(* IEC 61131-3 sources: ics/BLR1_PhoenixContact/BLR1_AXC1050_21/LogicalPOUs/MTR, 6 files *)

(* ---- MotorFB.ST ---- *)
(*@PROPERTIES_EX@
TYPE: POU
LOCALE: 0
IEC_LANGUAGE: ST
PLC_TYPE: independent
PROC_TYPE: independent
GROUP: MTRS.FB
*)
(*@KEY@:DESCRIPTION*)

(*@KEY@:END_DESCRIPTION*)
FUNCTION_BLOCK MotorFB

(*Group:Default*)

VAR_IN_OUT
    Mot_strct :	MTR;
    Aux_strct :	MTR_MISC;
END_VAR

VAR_INPUT
    Cycle :	CCL;
END_VAR

VAR_EXTERNAL
    TICK_1S_PLS :	BOOL;
END_VAR

VAR_OUTPUT
    Event :	MTR_EVENT;
END_VAR

(*@KEY@: WORKSHEET
NAME: MotorFB
IEC_LANGUAGE: ST
*)

IF TICK_1S_PLS and not Aux_strct.AuxFlag THEN
    Aux_strct.Tick_1S:= true;
END_IF;
Aux_strct.AuxFlag:= TICK_1S_PLS;

(*============================================================================*)
    (*Alarm Feedback processing*)
(*============================================================================*)
IF Mot_strct.CW.Enable and ((Aux_strct.COM and not Mot_strct.SW.RUN) or (not Aux_strct.COM and Mot_strct.SW.RUN)) THEN
    IF Aux_strct.Tick_1S THEN
        Aux_strct.AlrmTickCount:= Aux_strct.AlrmTickCount + 1;
    END_IF;
ELSE
    Aux_strct.AlrmTickCount:= 0;
END_IF;

IF Aux_strct.AlrmTickCount >= Aux_strct.SetOvertime THEN
    Aux_strct.AlarmFeedback:=true;
    Aux_strct.AlrmTickCount:= 0;
END_IF;

IF not Mot_strct.CW.ExtraEn and Aux_strct.COM THEN
    Aux_strct.AlarmBlock:= true;
END_IF;

Mot_strct.SW.AlarmAccum:= Aux_strct.AlarmFeedback or Mot_strct.CW.ExtraAlarm or Aux_strct.AlarmBlock;

IF Mot_strct.CW.ACK THEN
    Aux_strct.AlarmFeedback:=false;
    Aux_strct.AlarmBlock:= false;
END_IF;

(*============================================================================*)
    (*Auto/Manual mode selection*)
(*============================================================================*)
IF Mot_strct.CW.AutoMode THEN
    Mot_strct.SW.ManAuto:= true;
ELSIF Mot_strct.CW.ManMode THEN
    Mot_strct.SW.ManAuto:= false;
END_IF;

Mot_strct.SW.ManOK:= not Mot_strct.SW.AlarmAccum and Mot_strct.CW.AuxON and
    Mot_strct.CW.Enable and not Mot_strct.SW.ManAuto;
Mot_strct.SW.AutoOK:= not Mot_strct.SW.AlarmAccum and Mot_strct.CW.AuxON and
    Mot_strct.CW.Enable and Mot_strct.SW.ManAuto;

(*============================================================================*)
    (*Manual mode activation*)
(*============================================================================*)

IF Mot_strct.CW.ManStop or not Mot_strct.SW.ManOK THEN
    Mot_strct.SW.RunManual:=false;
ELSIF Mot_strct.CW.ManStart THEN
    Mot_strct.SW.RunManual:=true;
END_IF;

(*============================================================================*)
    (*Auto mode activation*)
(*============================================================================*)
Mot_strct.SW.RunAuto:= Mot_strct.SW.AutoOK and Cycle.SW.Running;

(*============================================================================*)
    (*Set command for start*)
(*============================================================================*)
Aux_strct.COM:=((Mot_strct.SW.RunManual and Mot_strct.SW.ManOK) or
    (Mot_strct.SW.RunAuto and Mot_strct.SW.AutoOK and Mot_strct.CW.AutoON));
Mot_strct.SW.COM:=Aux_strct.COM and not Mot_strct.CW.SimEn;

(*============================================================================*)
    (*Frequency limatation*)
(*============================================================================*)
Mot_strct.MaxFreq:= LIMIT(0.0, Mot_strct.MaxFreq, 50.0);
Mot_strct.MinFreq:= LIMIT(0.0, Mot_strct.MinFreq, Mot_strct.MaxFreq);
Mot_strct.ManFreq:= LIMIT(Mot_strct.MinFreq, Mot_strct.ManFreq, Mot_strct.MaxFreq);
Mot_strct.AutoFreq:= LIMIT(Mot_strct.MinFreq, Mot_strct.AutoFreq, Mot_strct.MaxFreq);

IF Mot_strct.SW.RunAuto and not Mot_strct.SW.AlarmAccum and Mot_strct.CW.AuxON THEN
    Aux_strct.SetValue:=Mot_strct.AutoFreq;
ELSIF not Mot_strct.SW.AlarmAccum and Mot_strct.SW.RunManual THEN
    Aux_strct.SetValue:=Mot_strct.ManFreq;
ELSE
    Aux_strct.SetValue:=0.0;
END_IF;

(*============================================================================*)
    (*Work time counter*)
(*============================================================================*)
IF Mot_strct.SW.COM and Aux_strct.Tick_1S THEN
    Aux_strct.Seconds:= Aux_strct.Seconds + udint#1;
END_IF;

Aux_strct.Minutes:= Aux_strct.Seconds / udint#60;
Aux_strct.Hours:= Aux_strct.Seconds / udint#3600;
Aux_strct.Days:= Aux_strct.Seconds / udint#86400;

(*============================================================================*)
    (*Aux time counters*)
(*============================================================================*)
IF Aux_strct.CT1_ON and Aux_strct.Tick_1S THEN
    Aux_strct.CT1:= Aux_strct.CT1 + 1;
ELSIF not Aux_strct.CT1_ON THEN
    Aux_strct.CT1:= 0;
END_IF;

IF Aux_strct.CT2_ON and Aux_strct.Tick_1S THEN
    Aux_strct.CT2:= Aux_strct.CT2 + 1;
ELSIF not Aux_strct.CT2_ON THEN
    Aux_strct.CT2:= 0;
END_IF;

(*============================================================================*)
    (*Status processing*)
(*============================================================================*)
IF Mot_strct.SW.AlarmAccum THEN                                                 (*Alarm*)
    Mot_strct.Status:=word#2;
ELSIF not Mot_strct.CW.ExtraEn THEN                                             (*Blocking*)
    Mot_strct.Status:=word#4;
ELSIF Mot_strct.SW.COM THEN                                                     (*Working*)
    Mot_strct.Status:=word#1;
ELSE                                                                            (*Stopped*)
    Mot_strct.Status:=word#0;
END_IF;

Mot_strct.CW.AutoMode:=false;
Mot_strct.CW.ManMode:=false;
Mot_strct.CW.ManStart:=false;
Mot_strct.CW.ManStop:=false;
Mot_strct.CW.ACK:=false;
Aux_strct.Tick_1S:= false;

(*============================================================================*)
(*Motor Pulse Events*)
(*============================================================================*)

Event.AlarmAccum:= false;
IF Mot_strct.SW.AlarmAccum and not Aux_strct.EVENT_1 THEN
    Event.AlarmAccum:= true;
    Aux_strct.EVENT_1:= true;
ELSIF not Mot_strct.SW.AlarmAccum THEN
    Aux_strct.EVENT_1:= false;
END_IF;
(*@KEY@: END_WORKSHEET *)
END_FUNCTION_BLOCK

(* ---- BLR_CTRL.ST ---- *)
(*@PROPERTIES_EX@
TYPE: POU
LOCALE: 0
IEC_LANGUAGE: ST
PLC_TYPE: independent
PROC_TYPE: independent
GROUP: MTRS
*)
(*@KEY@:DESCRIPTION*)

(*@KEY@:END_DESCRIPTION*)
PROGRAM BLR_CTRL

(*Group:Default*)

(*@KEY@: WORKSHEET
NAME: BLR_CTRL
IEC_LANGUAGE: ST
*)
(*@KEY@: END_WORKSHEET *)
END_PROGRAM

(* ---- MTR.ST ---- *)
(*@PROPERTIES_EX@
TYPE: POU
LOCALE: 0
IEC_LANGUAGE: ST
PLC_TYPE: independent
PROC_TYPE: independent
GROUP: MTRS
*)
(*@KEY@:DESCRIPTION*)

(*@KEY@:END_DESCRIPTION*)
PROGRAM MTR

(*Group:Default*)

VAR_EXTERNAL
    Cycle :	CCL;
    M :	MOTOR;
    WarnWord :	WRN;
    AI :	SENSOR;
END_VAR

VAR
    Pmp31FB :	MotorFB;
END_VAR

VAR_EXTERNAL
    M_AUX :	MOTOR_MISC;
END_VAR

VAR
    i :	INT;
    PmpsFB :	MotorFB;
END_VAR

VAR_EXTERNAL
    Blr11_BrnRun :	BOOL;
    Blr11_BrnFault :	BOOL;
    Blr12_BrnRun :	BOOL;
    Blr12_BrnFault :	BOOL;
    Blr13_BrnRun :	BOOL;
    Blr13_BrnFault :	BOOL;
    Blr21_BrnRun :	BOOL;
    Blr21_BrnFault :	BOOL;
    Blr22_BrnRun :	BOOL;
    Blr22_BrnFault :	BOOL;
END_VAR

VAR
    PumpsFB :	MotorFB;
    MB_TO_REAL :	MB_TO_REAL;
END_VAR

VAR_EXTERNAL
    SlvData_RSUNI_2 :	MBRTU_SlvData;
    SlvData_RSUNI_1 :	MBRTU_SlvData;
    MBTCP_Data :	MB_TCP_ARR_W_0_7167;
END_VAR

VAR
    j :	INT;
    j2 :	INT;
    j3 :	INT;
    j4 :	INT;
    j5 :	INT;
    j6 :	INT;
    j7 :	INT;
    REAL_TO_MB :	REAL_TO_MB;
    BoilersFB :	MotorFB;
    BlrCycle :	CCL;
END_VAR

VAR_EXTERNAL
    CCL :	CYCLE;
    Blr11_EmergCirc :	BOOL;
    Blr12_EmergCirc :	BOOL;
    Blr13_EmergCirc :	BOOL;
    Blr21_EmergCirc :	BOOL;
    Blr22_EmergCirc :	BOOL;
END_VAR

VAR
    MotorFB_1 :	MotorFB;
END_VAR

VAR_EXTERNAL
    M_EVENT :	MOTOR_EVENT;
END_VAR

(*@KEY@: WORKSHEET
NAME: MTR
IEC_LANGUAGE: ST
*)
Cycle.CW.AuxON:= true;
BlrCycle.SW.Running:= true;

FOR i:= 0 TO 4 DO
    j:= i * 32 + 3940;
    MBTCP_Data[j].X5:= true;
    M[i].CW.Enable:= true;
    M[i].CW.ExtraEn:= true;
    M[i].CW.AuxON:= true;
    M_AUX[i].SetOvertime:= 3;
END_FOR;

(*============================================================================*)
    (*Boiler 1.1 DI*)
(*============================================================================*)
M[0].CW.AutoON:=Blr11_BrnRun;
M[0].SW.RUN:=Blr11_BrnRun;
M[0].CW.ExtraEn:=Blr11_EmergCirc;
M[0].CW.ExtraAlarm:=Blr11_BrnFault;

(*============================================================================*)
    (*Boiler 1.2 DI*)
(*============================================================================*)
M[1].CW.AutoON:=Blr12_BrnRun;
M[1].SW.RUN:=Blr12_BrnRun;
M[1].CW.ExtraEn:=Blr12_EmergCirc;
M[1].CW.ExtraAlarm:=Blr12_BrnFault;

(*============================================================================*)
    (*Boiler 1.3 DI*)
(*============================================================================*)
M[2].CW.AutoON:=Blr13_BrnRun;
M[2].SW.RUN:=Blr13_BrnRun;
M[2].CW.ExtraEn:=Blr13_EmergCirc;
M[2].CW.ExtraAlarm:=Blr13_BrnFault;

(*============================================================================*)
    (*Boiler 2.1 DI*)
(*============================================================================*)
M[3].CW.AutoON:=Blr21_BrnRun;
M[3].SW.RUN:=Blr21_BrnRun;
M[3].CW.ExtraEn:=Blr21_EmergCirc;
M[3].CW.ExtraAlarm:=Blr21_BrnFault;

(*============================================================================*)
    (*Boiler 2.2 DI*)
(*============================================================================*)
M[4].CW.AutoON:=Blr22_BrnRun;
M[4].SW.RUN:=Blr22_BrnRun;
M[4].CW.ExtraEn:=Blr22_EmergCirc;
M[4].CW.ExtraAlarm:=Blr22_BrnFault;

(*============================================================================*)
M[1].AutoFreq:=M[0].AutoFreq;
M[2].AutoFreq:=M[0].AutoFreq;
M[4].AutoFreq:=M[3].AutoFreq;
(*============================================================================*)
    (*Boilers FB processing*)
(*============================================================================*)
FOR i:= 0 TO 4 DO
    BoilersFB(Mot_strct:=M[i],Aux_strct:=M_AUX[i],Cycle:=BlrCycle);
    M[i]:=BoilersFB.Mot_strct;
    M_AUX[i]:=BoilersFB.Aux_strct;
END_FOR;

(*============================================================================*)
FOR i:= 5 TO 7 DO
    j:= i - 5;
(*============================================================================*)
    (*Pump 3.x structure parameters*)
(*============================================================================*)
    M[i].CW.Enable:=M[i].SW.Rem;
    M[i].CW.AuxON:=CCL[2].CW.AuxON ;
    M[i].CW.ExtraAlarm:=M_AUX[i].DryMoveFault or M_AUX[i].TempFault;
    M[i].CW.ExtraEn:=true;
    M[i].SW.RUN:=M_AUX[i].DirRun or M_AUX[i].FCRun;
    M_AUX[i].SetOvertime:=90;
(*============================================================================*)
    (*Pump 3.x FC parameters*)
(*============================================================================*)
    M[i].ActFreq:=word_to_real(SlvData_RSUNI_2[j][0]) / 10.0;
    M[i].Power:=word_to_real(SlvData_RSUNI_2[j][2]) / 1000.0;a
    M[i].Current:=word_to_real(SlvData_RSUNI_2[j][4]) / 100.0;
    M[i].HeatSinkTemp:=word_to_real(SlvData_RSUNI_2[j][6]);
    M[i].FC_StatusWord:=SlvData_RSUNI_2[j][8];
    M[i].FC_AlarmWord:=DW_TO_DWORD(SlvData_RSUNI_2[j][10],SlvData_RSUNI_2[j][11]);
    M[i].FC_WarnWord:=DW_TO_DWORD(SlvData_RSUNI_2[j][12],SlvData_RSUNI_2[j][13]);

    M[i].RunHours:=dword_to_real(DW_TO_DWORD(SlvData_RSUNI_2[j][14],SlvData_RSUNI_2[j][15]));
    M[i].kWhCount:=dword_to_real(DW_TO_DWORD(SlvData_RSUNI_2[j][16],SlvData_RSUNI_2[j][17]));

(*============================================================================*)
    (*Pumps 3.x FB processing*)
(*============================================================================*)
    PumpsFB(Mot_strct:=M[i],Aux_strct:=M_AUX[i],Cycle:=CCL[2]);
    M[i]:=PumpsFB.Mot_strct;
    M_AUX[i]:=PumpsFB.Aux_strct;
    M_EVENT[i]:=PumpsFB.Event;
END_FOR;

(*============================================================================*)
FOR i:= 8 TO 10 DO
    j:= i - 8;
(*============================================================================*)
    (*Pump 5.x structure parameters*)
(*============================================================================*)
    M[i].CW.Enable:= M[i].SW.Rem;
    M[i].CW.AuxON:= Cycle.CW.AuxON;
    M[i].CW.ExtraAlarm:= M_AUX[i].DryMoveFault or M_AUX[i].TempFault;
    M[i].CW.ExtraEn:= true;
    M[i].SW.RUN:= M_AUX[i].DirRun or M_AUX[i].FCRun;
    M_AUX[i].SetOvertime:= 90;
(*============================================================================*)
    (*Pump 5.x FC parameters*)
(*============================================================================*)
    M[i].ActFreq:=word_to_real(SlvData_RSUNI_1[j][0]) / 10.0;
    M[i].Power:=word_to_real(SlvData_RSUNI_1[j][3]) / 100.0;
    M[i].Current:=word_to_real(SlvData_RSUNI_1[j][5]) / 100.0;
    M[i].HeatSinkTemp:=word_to_real(SlvData_RSUNI_1[j][6]);
    M[i].FC_StatusWord:=SlvData_RSUNI_1[j][8];
    M[i].FC_AlarmWord:=DW_TO_DWORD(SlvData_RSUNI_1[j][10],SlvData_RSUNI_1[j][11]);
    M[i].FC_WarnWord:=DW_TO_DWORD(SlvData_RSUNI_1[j][12],SlvData_RSUNI_1[j][13]);

    M[i].RunHours:=dword_to_real(DW_TO_DWORD(SlvData_RSUNI_1[j][14],SlvData_RSUNI_1[j][15]));
    M[i].kWhCount:=dword_to_real(DW_TO_DWORD(SlvData_RSUNI_1[j][16],SlvData_RSUNI_1[j][17]));

(*============================================================================*)
    (*Pumps 5.x FB processing*)
(*============================================================================*)
    PumpsFB(Mot_strct:=M[i],Aux_strct:=M_AUX[i],Cycle:=CCL[3]);
    M[i]:=PumpsFB.Mot_strct;
    M_AUX[i]:=PumpsFB.Aux_strct;
    M_EVENT[i]:=PumpsFB.Event;
END_FOR;

(*============================================================================*)
FOR i:= 11 TO 12 DO
    j:= i - 8;
(*============================================================================*)
    (*Pump 6.x structure parameters*)
(*============================================================================*)
    M[i].CW.Enable:=M[i].SW.Rem;
    M[i].CW.AuxON:=Cycle.CW.AuxON;
    M[i].CW.ExtraAlarm:=M_AUX[i].DryMoveFault or M_AUX[i].TempFault;
    M[i].CW.ExtraEn:=true;
    M[i].SW.RUN:=M_AUX[i].DirRun or M_AUX[i].FCRun;
    M_AUX[i].SetOvertime:=90;
(*============================================================================*)
    (*Pump 6.x FC parameters*)
(*============================================================================*)
    M[i].ActFreq:=word_to_real(SlvData_RSUNI_2[j][0]) / 10.0;
    M[i].Power:=word_to_real(SlvData_RSUNI_2[j][2]) / 1000.0;
    M[i].Current:=word_to_real(SlvData_RSUNI_2[j][4]) / 100.0;
    M[i].HeatSinkTemp:=word_to_real(SlvData_RSUNI_2[j][6]);
    M[i].FC_StatusWord:=SlvData_RSUNI_2[j][8];
    M[i].FC_AlarmWord:=DW_TO_DWORD(SlvData_RSUNI_2[j][10],SlvData_RSUNI_2[j][11]);
    M[i].FC_WarnWord:=DW_TO_DWORD(SlvData_RSUNI_2[j][12],SlvData_RSUNI_2[j][13]);

    M[i].RunHours:=dword_to_real(DW_TO_DWORD(SlvData_RSUNI_2[j][14],SlvData_RSUNI_2[j][15]));
    M[i].kWhCount:=dword_to_real(DW_TO_DWORD(SlvData_RSUNI_2[j][16],SlvData_RSUNI_2[j][17]));

(*============================================================================*)
    (*Pumps 6.x FB processing*)
(*============================================================================*)
    PumpsFB(Mot_strct:=M[i],Aux_strct:=M_AUX[i],Cycle:=CCL[4]);
    M[i]:=PumpsFB.Mot_strct;
    M_AUX[i]:=PumpsFB.Aux_strct;
    M_EVENT[i]:=PumpsFB.Event;
END_FOR;

(*============================================================================*)
    (*Reset CWs and rewrite parameters TO MB TCP*)
(*============================================================================*)
FOR i:= 5 TO 12 DO
    j:= i * 32 + 3940;
    j2:= j + 2;
    j3:= j + 3;
    j4:= j + 4;
    j5:= j + 5;
    j6:= j + 6;
    j7:= j + 7;

    REAL_TO_MB(IN:=M[i].MinFreq);
    MBTCP_Data[j2]:=REAL_TO_MB.LoWord;
    MBTCP_Data[j3]:=REAL_TO_MB.HiWord;

    REAL_TO_MB(IN:=M[i].MaxFreq);
    MBTCP_Data[j4]:=REAL_TO_MB.LoWord;
    MBTCP_Data[j5]:=REAL_TO_MB.HiWord;

    REAL_TO_MB(IN:=M[i].ManFreq);
    MBTCP_Data[j6]:=REAL_TO_MB.LoWord;
    MBTCP_Data[j7]:=REAL_TO_MB.HiWord;
END_FOR;

(*============================================================================*)
(*@KEY@: END_WORKSHEET *)
END_PROGRAM

(* ---- MTR3_CTRL.ST ---- *)
(*@PROPERTIES_EX@
TYPE: POU
LOCALE: 0
IEC_LANGUAGE: ST
PLC_TYPE: independent
PROC_TYPE: independent
GROUP: MTRS
*)
(*@KEY@:DESCRIPTION*)

(*@KEY@:END_DESCRIPTION*)
PROGRAM MTR3_CTRL

(*Group:Default*)

VAR
    RunPmpNum :	INT;
    TmpWTMax :	UDINT;
    TmpWTMin :	UDINT;
    TmpIndMax :	INT;
    TmpIndMin :	INT;
    i :	INT;
    StartPmpReq :	BOOL;
    StopPmpReq :	BOOL;
    Stage :	INT;
END_VAR

VAR_EXTERNAL
    CCL :	CYCLE;
END_VAR

VAR
    StartReqTmr :	TON;
    StopReqTmr :	TON;
    OverClckTmr :	TON;
    ReleaseTmr :	TON;
    TmpFreq :	REAL;
END_VAR

VAR_EXTERNAL
    M :	MOTOR;
    RGLTR :	REGULATOR;
    M_AUX :	MOTOR_MISC;
    MBTCP_Data :	MB_TCP_ARR_W_0_7167;
    AI :	SENSOR;
END_VAR

VAR
    MainPID :	FPID;
    TmpRotation :	BOOL;
    j :	INT;
END_VAR

VAR_EXTERNAL
    M_EVENT :	MOTOR_EVENT;
END_VAR

VAR
    TmpPmpAlarm :	BOOL;
    SysNum :	INT;
    LoInd :	INT;
    HiInd :	INT;
END_VAR

(*@KEY@: WORKSHEET
NAME: MTR3_CTRL
IEC_LANGUAGE: ST
*)
(*============================================================================*)
(*Work time sorting*)
(*Number of working pumps evaluation*)
(*PID min and max limits determination*)
(*============================================================================*)
SysNum:= 2;                                                                     (*Sequence number of cycle in cycles array (regulator in reg. array)*)
LoInd:= 5;                                                                      (*First number of pump in pumps array used here*)
HiInd:= 7;                                                                      (*Last number of pump in pumps array used here*)
RunPmpNum:= 0;
RGLTR[SysNum].LL:= 50.0;
RGLTR[SysNum].LH:= 0.0;

(*============================================================================*)
FOR i:= LoInd TO HiInd DO

    IF  M[i].SW.AutoOK and M[i].SW.RUN THEN                                     (*Working pump number determination*)
        RunPmpNum:= RunPmpNum + 1;

        IF  M[i].MaxFreq > RGLTR[SysNum].LH  THEN                               (*Assign pumps max. freq TO RGLTR. hight limit*)
            RGLTR[SysNum].LH:= M[i].MaxFreq;
        END_IF;

        IF  M[i].MinFreq < RGLTR[SysNum].LL THEN                                (*Assign pumps min. freq TO RGLTR. low limit*)
            RGLTR[SysNum].LL:= M[i].MinFreq;
        END_IF;
    END_IF;

    IF  not M[i].SW.AutoOK THEN                                                 (*Reset auto command IF  not auto*)
        M[i].CW.AutoON:= false;
    END_IF;

    M[i].AutoFreq:= RGLTR[SysNum].Y / 10.0;                                     (*Assign pumps min. freq TO RGLTR. low limit*)

(*============================================================================*)
    (*Pumps Dry motion*)
(*============================================================================*)
    j:= i * 3 + 31;

    M_AUX[i].CT1_ON:= (AI[j].RealValue <= 0.5) and M[i].SW.RUN and
        not M_AUX[i].DryMoveFault;

    IF  M_AUX[i].CT1 > 5 THEN
        M_AUX[i].DryMoveFault:= true;
    END_IF;

    M_AUX[i].CT2_ON:= (AI[j].RealValue >= 1.0) and M_AUX[i].DryMoveFault;

    IF  M_AUX[i].CT2 > 60 THEN
        M_AUX[i].DryMoveFault:= false;
    END_IF;

(*============================================================================*)
    (*Alarm action*)
(*============================================================================*)
    IF  M[i].SW.ManAuto and M_EVENT[i].AlarmAccum THEN
        TmpPmpAlarm:= true;
    END_IF;
END_FOR;
(*============================================================================*)

(*============================================================================*)
    (*Set rotation command*)
(*============================================================================*)
IF  CCL[SysNum].CW.Rotation THEN
    CCL[SysNum].SW.RotationON:= true;
    CCL[SysNum].CW.Rotation:= false;
END_IF;

(*============================================================================*)
    (*Start/Stop conditions*)
(*============================================================================*)
StartReqTmr(IN:=(((RGLTR[SysNum].Y / 10.0) >= (RGLTR[SysNum].LH - 1.0)) and
    (RGLTR[SysNum].ActVal < RGLTR[SysNum].SP) and not StartPmpReq and
    CCL[SysNum].SW.Running),PT:=t#60s);                                         (*Start auxiliary pump condition*)

StopReqTmr(IN:=(((RGLTR[SysNum].Y / 10.0) <= (RGLTR[SysNum].LL + 1.0)) and
    (RGLTR[SysNum].ActVal >= RGLTR[SysNum].SP) and not StopPmpReq and
    CCL[SysNum].SW.Running),PT:=t#60s);                                         (*Stop pump condition*)

(*============================================================================*)
    (*Cycle handling*)
(*============================================================================*)
IF  CCL[SysNum].SW.Running THEN
    IF  (StartReqTmr.Q or (RunPmpNum < 1) or TmpPmpAlarm) and (Stage = 0) THEN  (*Stage route: 1 >> 2 >> 0*)
        Stage:= 1;
        IF  TmpPmpAlarm THEN
            TmpPmpAlarm:= false;
        END_IF;
    ELSIF  CCL[SysNum].SW.RotationON and (RunPmpNum > 0) and (Stage = 0) THEN   (*Stage route: 3 >> 1 >> 2 >> 4 >> 0*)
        TmpRotation:= true;
        Stage:= 3;
    ELSIF  StopReqTmr.Q and (Stage = 0) THEN                                    (*Stage route: 3 >> 4 >> 0*)
        Stage:= 3;
    END_IF;
ELSE
    StartPmpReq:= false;
    StopPmpReq:= false;
    TmpFreq:= 0.0;
    CCL[SysNum].SW.RotationON:= false;
    TmpRotation:= false;
    Stage:= 0;
    TmpPmpAlarm:= false;

    FOR i:= LoInd TO HiInd DO
        M[i].CW.AutoON:= false;
    END_FOR;
END_IF;

OverClckTmr(IN:=StartPmpReq and not OverClckTmr.Q,PT:=t#3s);                    (*Overclocking pulse timer*)
ReleaseTmr(IN:=StopPmpReq and not ReleaseTmr.Q,PT:=t#3s);                       (*Releasing pulse timer*)

CASE Stage OF

    0:	StartPmpReq:= false;
        StopPmpReq:= false;
        TmpPmpAlarm:= false;
        CCL[SysNum].SW.RotationON:= false;
        TmpRotation:= false;
        TmpFreq:= 0.0;

    1:	StartPmpReq:= true;                                                     (*Determ. higher work time*)
        TmpWTMin:= udint#0;
        TmpIndMin:= 0;
        FOR i:= LoInd TO HiInd DO
            IF  M_AUX[i].Seconds >= TmpWTMin THEN
                TmpWTMin:= M_AUX[i].Seconds;                                    (*Assign. higher work time TO temporary var.*)
            END_IF;
        END_FOR;

        FOR i:= LoInd TO HiInd DO
            IF  M[i].SW.AutoOK and not M[i].SW.RUN THEN                         (*Determ. lowest work time pump*)
                IF  M_AUX[i].Seconds <= TmpWTMin THEN
                    TmpWTMin:= M_AUX[i].Seconds;
                    TmpIndMin:= i;                                              (*Determ. lowest work time pump index*)
                END_IF;
            END_IF;
        END_FOR;
        IF  (TmpIndMin < LoInd) and (TmpIndMin > HiInd) THEN
            Stage:= 5;
        ELSE
            M[TmpIndMin].CW.AutoON:= true;                                      (*Start lowest work time pump*)
            TmpFreq:= M[TmpIndMin].MinFreq;                                     (*with min. frequency*)
            Stage:= 2;
        END_IF;

    2:	M[TmpIndMin].AutoFreq:= TmpFreq;                                        (*Overclocking new pump*)
        IF  OverClckTmr.Q THEN
            TmpFreq:= TmpFreq + 1.0;
        ELSIF  M[TmpIndMin].AutoFreq >= (RGLTR[SysNum].Y / 10.0)  THEN
            StartPmpReq:= false;
            IF  TmpRotation THEN
                Stage:= 4;
            ELSE
                Stage:= 5;
            END_IF;
        END_IF;

    3:	TmpWTMax:= udint#0;                                                     (*Determ. highest work time pump*)
        TmpIndMax:= 0;
        FOR i:= LoInd TO HiInd DO
            IF  M[i].SW.AutoOK and M[i].SW.RUN THEN
                IF  M_AUX[i].Seconds >= TmpWTMax THEN
                    TmpWTMax:= M_AUX[i].Seconds;
                    TmpIndMax:= i;
                END_IF;
            END_IF;
        END_FOR;
        IF  TmpRotation THEN
            Stage:= 1;
        ELSE
            TmpFreq:= RGLTR[SysNum].Y / 10.0;
            Stage:= 4;
        END_IF;

    4:	StopPmpReq:= true;                                                      (*Releasing highest work time pump*)
        M[TmpIndMax].AutoFreq:= TmpFreq;
        IF  ReleaseTmr.Q THEN
            TmpFreq:= TmpFreq - 1.0;
        ELSIF  M[TmpIndMax].AutoFreq <= M[TmpIndMax].MinFreq THEN
            M[TmpIndMax].CW.AutoON:= false;
            StopPmpReq:= false;
            Stage:= 5;
            TmpFreq:= 0.0;
        END_IF;

    5:	StartPmpReq:= false;
        StopPmpReq:= false;
        TmpPmpAlarm:= false;
        CCL[SysNum].SW.RotationON:= false;
        TmpRotation:= false;
        TmpFreq:= 0.0;
        Stage:= 0;
END_CASE;

(*============================================================================*)
    (*Main PID*)
(*============================================================================*)
RGLTR[SysNum].ActVal:= AI[55].RealValue - AI[45].RealValue;
MainPID(REMOTE:=CCL[SysNum].SW.Running,
        AUTO:=true,
        DIRECTN:=false,
        INTLCK:=(RunPmpNum <= 0),
        Tscan:=1.0,
        Yman:=RGLTR[SysNum].ManVal,
        SPR:=(RGLTR[SysNum].SP * 100.0),
        SPL:=0.0,
        X:=(RGLTR[SysNum].ActVal * 100.0),
        KP:=RGLTR[SysNum].Kp,
        TI:=RGLTR[SysNum].Tn,
        TD:=RGLTR[SysNum].Tv,
        HIGH:=(RGLTR[SysNum].LH * 10.0),
        LOW:=(RGLTR[SysNum].LL * 10.0),
        INTLCKV:=0.0);
RGLTR[SysNum].Y:=MainPID.Yout;

(*============================================================================*)
(*@KEY@: END_WORKSHEET *)
END_PROGRAM

(* ---- MTR5_CTRL.ST ---- *)
(*@PROPERTIES_EX@
TYPE: POU
LOCALE: 0
IEC_LANGUAGE: ST
PLC_TYPE: independent
PROC_TYPE: independent
GROUP: MTRS
*)
(*@KEY@:DESCRIPTION*)

(*@KEY@:END_DESCRIPTION*)
PROGRAM MTR5_CTRL

(*Group:Default*)

VAR
    RunPmpNum :    INT;
    TmpWTMax :    UDINT;
    TmpWTMin :    UDINT;
    TmpIndMax :    INT;
    TmpIndMin :    INT;
    i :    INT;
    StartPmpReq :    BOOL;
    StopPmpReq :    BOOL;
    Stage :    INT;
END_VAR

VAR_EXTERNAL
    CCL :    CYCLE;
END_VAR

VAR
    StartReqTmr :    TON;
    StopReqTmr :    TON;
    OverClckTmr :    TON;
    ReleaseTmr :    TON;
    TmpFreq :    REAL;
END_VAR

VAR_EXTERNAL
    M :    MOTOR;
    RGLTR :    REGULATOR;
    M_AUX :    MOTOR_MISC;
    MBTCP_Data :    MB_TCP_ARR_W_0_7167;
    AI :    SENSOR;
END_VAR

VAR
    MainPID :    FPID;
    TmpRotation :    BOOL;
    j :    INT;
END_VAR

VAR_EXTERNAL
    M_EVENT :    MOTOR_EVENT;
END_VAR

VAR
    TmpPmpAlarm :    BOOL;
    SysNum :    INT;
    LoInd :    INT;
    HiInd :    INT;
END_VAR

(*@KEY@: WORKSHEET
NAME: MTR5_CTRL
IEC_LANGUAGE: ST
*)
(*============================================================================*)
(*Work time sorting*)
(*Number of working pumps evaluation*)
(*PID min and max limits determination*)
(*============================================================================*)
SysNum:= 3;                                                                     (*Sequence number of cycle in cycles array (regulator in reg. array)*)
LoInd:= 8;                                                                      (*First number of pump in pumps array used here*)
HiInd:= 10;                                                                     (*Last number of pump in pumps array used here*)
RunPmpNum:= 0;
RGLTR[SysNum].LL:= 50.0;
RGLTR[SysNum].LH:= 0.0;

(*============================================================================*)
FOR i:= LoInd TO HiInd do

    IF M[i].SW.AutoOK and M[i].SW.RUN THEN                                      (*Working pump number determination*)
        RunPmpNum:= RunPmpNum + 1;

        IF M[i].MaxFreq > RGLTR[SysNum].LH  THEN                                (*Assign pumps max. freq TO RGLTR. hight limit*)
            RGLTR[SysNum].LH:= M[i].MaxFreq;
        END_IF;

        IF M[i].MinFreq < RGLTR[SysNum].LL THEN                                 (*Assign pumps min. freq TO RGLTR. low limit*)
            RGLTR[SysNum].LL:= M[i].MinFreq;
        END_IF;
    END_IF;

    IF not M[i].SW.AutoOK THEN                                                  (*Reset auTO command IF not auto*)
        M[i].CW.AutoON:= false;
    END_IF;

    M[i].AutoFreq:= RGLTR[SysNum].Y / 10.0;                                      (*Assign pumps min. freq TO RGLTR. low limit*)

(*============================================================================*)
    (*Pumps Dry motion*)
(*============================================================================*)
    j:= i * 2 - 16;

    M_AUX[i].CT1_ON:= (AI[j].RealValue <= 0.5) and M[i].SW.RUN and not M_AUX[i].DryMoveFault;

    IF M_AUX[i].CT1 > 5 THEN
        M_AUX[i].DryMoveFault:= true;
    END_IF;

    M_AUX[i].CT2_ON:= (AI[j].RealValue >= 1.0) and M_AUX[i].DryMoveFault;

    IF M_AUX[i].CT2 > 60 THEN
        M_AUX[i].DryMoveFault:= false;
    END_IF;

(*============================================================================*)
    (*Alarm action*)
(*============================================================================*)
    IF M[i].SW.ManAuTO and M_EVENT[i].AlarmAccum THEN
        TmpPmpAlarm:= true;
    END_IF;
END_FOR;
(*============================================================================*)

(*============================================================================*)
    (*Set rotation command*)
(*============================================================================*)
IF CCL[SysNum].CW.Rotation THEN
    CCL[SysNum].SW.RotationON:= true;
    CCL[SysNum].CW.Rotation:= false;
END_IF;

(*============================================================================*)
    (*Start/Stop conditions*)
(*============================================================================*)
StartReqTmr(IN:=(((RGLTR[SysNum].Y / 10.0) >= (RGLTR[SysNum].LH - 2.0)) and
    (RGLTR[SysNum].ActVal < RGLTR[SysNum].SP) and not StartPmpReq and
    CCL[SysNum].SW.Running),PT:=t#60s);                                         (*Start auxiliary pump condition*)

StopReqTmr(IN:=(((RGLTR[SysNum].Y / 10.0) <= (RGLTR[SysNum].LL + 1.0)) and
    RGLTR[SysNum].ActVal >= RGLTR[SysNum].SP) and not StopPmpReq and
    CCL[SysNum].SW.Running),PT:=t#60s);                                         (*Stop pump condition*)

(*============================================================================*)
    (*Cycle handling*)
(*============================================================================*)
IF CCL[SysNum].SW.Running THEN
    IF (StartReqTmr.Q or (RunPmpNum < 1) or TmpPmpAlarm) and (Stage = 0) THEN   (*Stage route: 1 >> 2 >> 5 >> 0*)
        Stage:= 1;
        IF TmpPmpAlarm THEN
            TmpPmpAlarm:= false;
        END_IF;
    ELSIF CCL[SysNum].SW.RotationON and (RunPmpNum > 0) and (Stage = 0) THEN    (*Stage route: 3 >> 1 >> 2 >> 4 >> 5 >> 0*)
        TmpRotation:= true;
        Stage:= 3;
    ELSIF StopReqTmr.Q and (Stage = 0) THEN                                     (*Stage route: 3 >> 4 >> 5 >> 0*)
        Stage:= 3;
    END_IF;
ELSE
    StartPmpReq:= false;
    StopPmpReq:= false;
    TmpFreq:= 0.0;
    CCL[3].SW.RotationON:= false;
    TmpRotation:= false;
    Stage:= 0;
    TmpPmpAlarm:= false;

    FOR i:= LoInd TO HiInd do
        M[i].CW.AutoON:= false;
    END_FOR;
END_IF;

OverClckTmr(IN:=StartPmpReq and not OverClckTmr.Q,PT:=t#3s);                    (*Overclocking pulse timer*)
ReleaseTmr(IN:=StopPmpReq and not ReleaseTmr.Q,PT:=t#3s);                       (*Releasing pulse timer*)

CASE Stage OF

    0:  StartPmpReq:= false;
        StopPmpReq:= false;
        TmpPmpAlarm:= false;
        CCL[3].SW.RotationON:= false;
        TmpRotation:= false;
        TmpFreq:= 0.0;

    1:  StartPmpReq:= true;                                                     (*Determ. higher work time*)
        TmpWTMin:= udint#0;
        TmpIndMin:= 0;
        FOR i:= LoInd TO HiInd do
            IF M_AUX[i].Seconds >= TmpWTMin THEN
                TmpWTMin:= M_AUX[i].Seconds;                                    (*Assign. higher work time TO temporary var.*)
            END_IF;
        END_FOR;

        FOR i:= LoInd TO HiInd do
            IF M[i].SW.AutoOK and not M[i].SW.RUN THEN                          (*Determ. lowest work time pump*)
                IF M_AUX[i].Seconds <= TmpWTMin THEN
                    TmpWTMin:= M_AUX[i].Seconds;
                    TmpIndMin:= i;                                              (*Determ. lowest work time pump index*)
                END_IF;
            END_IF;
        END_FOR;
        IF (TmpIndMin < LoInd) and (TmpIndMin > HiInd) THEN
            Stage:= 5;
        ELSE
            M[TmpIndMin].CW.AutoON:= true;                                      (*Start lowest work time pump*)
            TmpFreq:= M[TmpIndMin].MinFreq;                                     (*with min. frequency*)
            Stage:= 2;
        END_IF;

    2:  M[TmpIndMin].AutoFreq:= TmpFreq;                                        (*Overclocking new pump*)
        IF OverClckTmr.Q THEN
            TmpFreq:= TmpFreq + 1.0;
        ELSIF M[TmpIndMin].AutoFreq >= (RGLTR[SysNum].Y / 10.0)  THEN
            StartPmpReq:= false;
            IF TmpRotation THEN
                Stage:= 4;
            ELSE
                Stage:= 5;
            END_IF;
        END_IF;

    3:  TmpWTMax:= udint#0;                                                     (*Determ. highest work time pump*)
        TmpIndMax:= 0;
        FOR i:= LoInd TO HiInd DO
            IF M[i].SW.AutoOK and M[i].SW.RUN THEN
                IF M_AUX[i].Seconds >= TmpWTMax THEN
                    TmpWTMax:= M_AUX[i].Seconds;
                    TmpIndMax:= i;
                END_IF;
            END_IF;
        END_FOR;
        IF TmpRotation THEN
            Stage:= 1;
        ELSE
            TmpFreq:= RGLTR[SysNum].Y / 10.0;
            Stage:= 4;
        END_IF;

    4:  StopPmpReq:= true;                                                      (*Releasing highest work time pump*)
        M[TmpIndMax].AutoFreq:= TmpFreq;
        IF ReleaseTmr.Q THEN
            TmpFreq:= TmpFreq - 1.0;
        ELSIF M[TmpIndMax].AutoFreq <= M[TmpIndMax].MinFreq THEN
            M[TmpIndMax].CW.AutoON:= false;
            StopPmpReq:= false;
            Stage:= 5;
            TmpFreq:= 0.0;
        END_IF;

    5:  StartPmpReq:= false;
        StopPmpReq:= false;
        TmpPmpAlarm:= false;
        CCL[SysNum].SW.RotationON:= false;
        TmpRotation:= false;
        TmpFreq:= 0.0;
        Stage:= 0;
END_CASE;

(*============================================================================*)
    (*Main PID*)
(*============================================================================*)
RGLTR[SysNum].ActVal:= AI[7].RealValue - AI[6].RealValue;
MainPID(REMOTE:=CCL[SysNum].SW.Running,
        AUTO:=true,
        DIRECTN:=false,
        INTLCK:=(RunPmpNum <= 0),
        Tscan:=1.0,
        Yman:=RGLTR[SysNum].ManVal,
        SPR:=(RGLTR[SysNum].SP * 100.0),
        SPL:=0.0,
        X:=(RGLTR[SysNum].ActVal * 100.0),
        KP:=RGLTR[SysNum].Kp,
        TI:=RGLTR[SysNum].Tn,
        TD:=RGLTR[SysNum].Tv,
        HIGH:=(RGLTR[SysNum].LH * 10.0),
        LOW:=(RGLTR[SysNum].LL * 10.0),
        INTLCKV:=0.0);
RGLTR[SysNum].Y:=MainPID.Yout;

(*============================================================================*)

(*@KEY@: END_WORKSHEET *)
END_PROGRAM

(* ---- MTR6_CTRL.ST ---- *)
(*@PROPERTIES_EX@
TYPE: POU
LOCALE: 0
IEC_LANGUAGE: ST
PLC_TYPE: independent
PROC_TYPE: independent
GROUP: MTRS
*)
(*@KEY@:DESCRIPTION*)

(*@KEY@:END_DESCRIPTION*)
PROGRAM MTR6_CTRL

(*Group:Default*)

VAR
    RunPmpNum :    INT;
    TmpWTMax :    UDINT;
    TmpWTMin :    UDINT;
    TmpIndMax :    INT;
    TmpIndMin :    INT;
    i :    INT;
    StartPmpReq :    BOOL;
    STOpPmpReq :    BOOL;
    Stage :    INT;
END_VAR

VAR_EXTERNAL
    CCL :    CYCLE;
END_VAR

VAR
    StartReqTmr :    TON;
    STOpReqTmr :    TON;
    OverClckTmr :    TON;
    ReleaseTmr :    TON;
    TmpFreq :    REAL;
END_VAR

VAR_EXTERNAL
    M :    MOTOR;
    RGLTR :    REGULATOR;
    M_AUX :    MOTOR_MISC;
    MBTCP_Data :    MB_TCP_ARR_W_0_7167;
    AI :    SENSOR;
END_VAR

VAR
    MainPID :    FPID;
    TmpRotation :    BOOL;
    j :    INT;
END_VAR

VAR_EXTERNAL
    M_EVENT :    MOTOR_EVENT;
END_VAR

VAR
    TmpPmpAlarm :    BOOL;
    SysNum :    INT;
    LoInd :    INT;
    HiInd :    INT;
END_VAR

(*@KEY@: WORKSHEET
NAME: MTR6_CTRL
IEC_LANGUAGE: ST
*)
(*============================================================================*)
(*Work time sorting*)
(*Number of working pumps evaluation*)
(*PID min and max limits determination*)
(*============================================================================*)
SysNum:= 4;                                                                     (*Sequence number of cycle in cycles array (regulaTOr in reg. array)*)
LoInd:= 11;                                                                     (*First number of pump in pumps array used here*)
HiInd:= 12;                                                                     (*Last number of pump in pumps array used here*)
RunPmpNum:= 0;
RGLTR[SysNum].LL:= 50.0;
RGLTR[SysNum].LH:= 0.0;

(*============================================================================*)
FOR i:= LoInd TO HiInd DO

    IF M[i].SW.AuTOOK and M[i].SW.RUN THEN                                       (*Working pump number determination*)
        RunPmpNum:= RunPmpNum + 1;

        IF M[i].MaxFreq > RGLTR[SysNum].LH  THEN                                (*Assign pumps max. freq TO RGLTR. hight limit*)
            RGLTR[SysNum].LH:= M[i].MaxFreq;
        END_IF;

        IF M[i].MinFreq < RGLTR[SysNum].LL THEN                                 (*Assign pumps min. freq TO RGLTR. low limit*)
            RGLTR[SysNum].LL:= M[i].MinFreq;
        END_IF;
    END_IF;

    IF not M[i].SW.AuTOOK THEN                                                  (*Reset auTO command IF not auTO*)
        M[i].CW.AuTOON:= false;
    END_IF;

    M[i].AuTOFreq:= RGLTR[SysNum].Y / 10.0;                                     (*Assign pumps min. freq TO RGLTR. low limit*)

(*============================================================================*)
(*Pumps Dry motion*)
(*============================================================================*)

    M_AUX[i].CT1_ON:= (AI[70].RealValue <= 0.5) and M[i].SW.RUN and not M_AUX[i].DryMoveFault;

    IF M_AUX[i].CT1 > 5 THEN
        M_AUX[i].DryMoveFault:= true;
    END_IF;

    M_AUX[i].CT2_ON:= (AI[70].RealValue >= 1.0) and M_AUX[i].DryMoveFault;

    IF M_AUX[i].CT2 > 60 THEN
        M_AUX[i].DryMoveFault:= false;
    END_IF;

(*============================================================================*)
(*Alarm action*)
(*============================================================================*)
    IF M[i].SW.ManAuTO and M_EVENT[i].AlarmAccum THEN
        TmpPmpAlarm:= true;
    END_IF;
END_FOR;
(*============================================================================*)

(*============================================================================*)
(*Set rotation command*)
(*============================================================================*)
IF CCL[SysNum].CW.Rotation THEN
    CCL[SysNum].SW.RotationON:= true;
    CCL[SysNum].CW.Rotation:= false;
END_IF;

(*============================================================================*)
(*Start/STOp conditions*)
(*============================================================================*)
StartReqTmr(IN:=(((RGLTR[SysNum].Y / 10.0) >= (RGLTR[SysNum].LH - 1.0)) and
    (RGLTR[SysNum].ActVal < RGLTR[SysNum].SP) and not StartPmpReq and
    CCL[SysNum].SW.Running),PT:=t#60s);                                         (*Start auxiliary pump condition*)

STOpReqTmr(IN:=(((RGLTR[SysNum].Y / 10.0) <= (RGLTR[SysNum].LL + 1.0)) and
	(RGLTR[SysNum].ActVal >= RGLTR[SysNum].SP) and not STOpPmpReq and
	CCL[SysNum].SW.Running),PT:=t#60s);    										(*STOp pump condition*)

(*============================================================================*)
(*Cycle handling*)
(*============================================================================*)
IF CCL[SysNum].SW.Running THEN
    IF (StartReqTmr.Q or (RunPmpNum < 1) or TmpPmpAlarm) and (Stage = 0) THEN   (*Stage route: 1 >> 2 >> 0*)
        Stage:= 1;
        IF TmpPmpAlarm THEN
            TmpPmpAlarm:= false;
        END_IF;
    elsIF CCL[SysNum].SW.RotationON and (RunPmpNum > 0) and (Stage = 0) THEN    (*Stage route: 3 >> 1 >> 2 >> 4 >> 0*)
        TmpRotation:= true;
        Stage:= 3;
    elsIF STOpReqTmr.Q and (Stage = 0) THEN                                     (*Stage route: 3 >> 4 >> 0*)
        Stage:= 3;
    END_IF;
else
    StartPmpReq:= false;
    STOpPmpReq:= false;
    TmpFreq:= 0.0;
    CCL[SysNum].SW.RotationON:= false;
    TmpRotation:= false;
    Stage:= 0;
    TmpPmpAlarm:= false;

    FOR i:= LoInd TO HiInd DO
        M[i].CW.AuTOON:= false;
    END_FOR;
END_IF;

OverClckTmr(IN:=StartPmpReq and not OverClckTmr.Q,PT:=t#3s);                    (*Overclocking pulse timer*)
ReleaseTmr(IN:=STOpPmpReq and not ReleaseTmr.Q,PT:=t#3s);                       (*Releasing pulse timer*)

CASE Stage OF

    0:  StartPmpReq:= false;
        STOpPmpReq:= false;
        TmpPmpAlarm:= false;
        CCL[SysNum].SW.RotationON:= false;
        TmpRotation:= false;
        TmpFreq:= 0.0;

    1:  StartPmpReq:= true;                                                     (*Determ. higher work time*)
        TmpWTMin:= udint#0;
        TmpIndMin:= 0;
        FOR i:= LoInd TO HiInd DO
            IF M_AUX[i].Seconds >= TmpWTMin THEN
                TmpWTMin:= M_AUX[i].Seconds;                                    (*Assign. higher work time TO temporary var.*)
            END_IF;
        END_FOR;

        FOR i:= LoInd TO HiInd DO
            IF M[i].SW.AuTOOK and not M[i].SW.RUN THEN                          (*Determ. lowest work time pump*)
                IF M_AUX[i].Seconds <= TmpWTMin THEN
                    TmpWTMin:= M_AUX[i].Seconds;
                    TmpIndMin:= i;                                              (*Determ. lowest work time pump index*)
                END_IF;
            END_IF;
        END_FOR;
        IF (TmpIndMin < LoInd) and (TmpIndMin > HiInd) THEN
            Stage:= 5;
        else
            M[TmpIndMin].CW.AuTOON:= true;                                      (*Start lowest work time pump*)
            TmpFreq:= M[TmpIndMin].MinFreq;                                     (*with min. frequency*)
            Stage:= 2;
        END_IF;

    2:  M[TmpIndMin].AuTOFreq:= TmpFreq;                                        (*Overclocking new pump*)
        IF OverClckTmr.Q THEN
            TmpFreq:= TmpFreq + 1.0;
        elsIF M[TmpIndMin].AuTOFreq >= (RGLTR[SysNum].Y / 10.0)  THEN
            StartPmpReq:= false;
            IF TmpRotation THEN
                Stage:= 4;
            else
                Stage:= 5;
            END_IF;
        END_IF;

    3:  TmpWTMax:= udint#0;                                                     (*Determ. highest work time pump*)
        TmpIndMax:= 0;
        FOR i:= LoInd TO HiInd DO
            IF M[i].SW.AuTOOK and M[i].SW.RUN THEN
                IF M_AUX[i].Seconds >= TmpWTMax THEN
                    TmpWTMax:= M_AUX[i].Seconds;
                    TmpIndMax:= i;
                END_IF;
            END_IF;
        END_FOR;
        IF TmpRotation THEN
            Stage:= 1;
        else
            TmpFreq:= RGLTR[SysNum].Y / 10.0;
            Stage:= 4;
        END_IF;

    4:  STOpPmpReq:= true; 		                                                (*Releasing highest work time pump*)
        M[TmpIndMax].AuTOFreq:= TmpFreq;
        IF ReleaseTmr.Q THEN
            TmpFreq:= TmpFreq - 1.0;
        elsIF M[TmpIndMax].AuTOFreq <= M[TmpIndMax].MinFreq THEN
            M[TmpIndMax].CW.AuTOON:= false;
            STOpPmpReq:= false;
            Stage:= 5;
            TmpFreq:= 0.0;
        END_IF;

    5:  StartPmpReq:= false;
        STOpPmpReq:= false;
        TmpPmpAlarm:= false;
        CCL[SysNum].SW.RotationON:= false;
        TmpRotation:= false;
        TmpFreq:= 0.0;
        Stage:= 0;
END_CASE;

(*============================================================================*)
(*Main PID*)
(*============================================================================*)
RGLTR[SysNum].ActVal:= AI[71].RealValue - AI[70].RealValue;
MainPID(REMOTE:=CCL[SysNum].SW.Running,
        AUTO:=true,
        DIRECTN:=false,
        INTLCK:=(RunPmpNum <= 0),
        Tscan:=1.0,
        Yman:=RGLTR[SysNum].ManVal,
        SPR:=(RGLTR[SysNum].SP * 100.0),
        SPL:=0.0,
        X:=(RGLTR[SysNum].ActVal * 100.0),
        KP:=RGLTR[SysNum].Kp,
        TI:=RGLTR[SysNum].Tn,
        TD:=RGLTR[SysNum].Tv,
        HIGH:=(RGLTR[SysNum].LH * 10.0),
        LOW:=(RGLTR[SysNum].LL * 10.0),
        INTLCKV:=0.0);
RGLTR[SysNum].Y:=MainPID.Yout;

(*============================================================================*)
(*@KEY@: END_WORKSHEET *)
END_PROGRAM
